Append3 := InternalAppend(destinationString, sources);
END_METHOD

METHOD Append4 : BOOL
VAR_INPUT
	destinationString : ANY_STRING;
	sourceString1 : WSTRING(255);
	sourceString2 : WSTRING(255);
	sourceString3 : WSTRING(255);
	sourceString4 : WSTRING(255);
END_VAR
VAR
	sources : ARRAY [1..4] OF POINTER TO WSTRING(255);
END_VAR
sources[1] := ADR(sourceString1);
sources[2] := ADR(sourceString2);
sources[3] := ADR(sourceString3);
sources[4] := ADR(sourceString4);

Append4 := InternalAppend(destinationString, sources);
END_METHOD

METHOD Append5 : BOOL
VAR_INPUT
	destinationString : ANY_STRING;
	sourceString1 : WSTRING(255);
	sourceString2 : WSTRING(255);
	sourceString3 : WSTRING(255);
	sourceString4 : WSTRING(255);
	sourceString5 : WSTRING(255);
END_VAR
VAR
	sources : ARRAY [1..5] OF POINTER TO WSTRING(255);
END_VAR
sources[1] := ADR(sourceString1);
sources[2] := ADR(sourceString2);
sources[3] := ADR(sourceString3);
sources[4] := ADR(sourceString4);
sources[5] := ADR(sourceString5);

Append5 := InternalAppend(destinationString, sources);
END_METHOD

METHOD Append6 : BOOL
VAR_INPUT
	destinationString : ANY_STRING;
	sourceString1 : WSTRING(255);
	sourceString2 : WSTRING(255);
	sourceString3 : WSTRING(255);
	sourceString4 : WSTRING(255);
	sourceString5 : WSTRING(255);
	sourceString6 : WSTRING(255);
END_VAR
VAR
	sources : ARRAY [1..6] OF POINTER TO WSTRING(255);
END_VAR
sources[1] := ADR(sourceString1);
sources[2] := ADR(sourceString2);
sources[3] := ADR(sourceString3);
sources[4] := ADR(sourceString4);
sources[5] := ADR(sourceString5);
sources[6] := ADR(sourceString6);

Append6 := InternalAppend(destinationString, sources);
END_METHOD

METHOD Append7 : BOOL
VAR_INPUT
	destinationString : ANY_STRING;
	sourceString1 : WSTRING(255);
	sourceString2 : WSTRING(255);
	sourceString3 : WSTRING(255);
	sourceString4 : WSTRING(255);
	sourceString5 : WSTRING(255);
	sourceString6 : WSTRING(255);
	sourceString7 : WSTRING(255);
END_VAR
VAR
	sources : ARRAY [1..7] OF POINTER TO WSTRING(255);
END_VAR
sources[1] := ADR(sourceString1);
sources[2] := ADR(sourceString2);
sources[3] := ADR(sourceString3);
sources[4] := ADR(sourceString4);
sources[5] := ADR(sourceString5);
sources[6] := ADR(sourceString6);
sources[7] := ADR(sourceString7);

Append7 := InternalAppend(destinationString, sources);
END_METHOD

METHOD Append8 : BOOL
VAR_INPUT
	destinationString : ANY_STRING;
	sourceString1 : WSTRING(255);
	sourceString2 : WSTRING(255);
	sourceString3 : WSTRING(255);
	sourceString4 : WSTRING(255);
	sourceString5 : WSTRING(255);
	sourceString6 : WSTRING(255);
	sourceString7 : WSTRING(255);
	sourceString8 : WSTRING(255);
END_VAR
VAR
	sources : ARRAY [1..8] OF POINTER TO WSTRING(255);
END_VAR
sources[1] := ADR(sourceString1);
sources[2] := ADR(sourceString2);
sources[3] := ADR(sourceString3);
sources[4] := ADR(sourceString4);
sources[5] := ADR(sourceString5);
sources[6] := ADR(sourceString6);
sources[7] := ADR(sourceString7);
sources[8] := ADR(sourceString8);

Append8 := InternalAppend(destinationString, sources);
END_METHOD

METHOD Append9 : BOOL
VAR_INPUT
	destinationString : ANY_STRING;
	sourceString1 : WSTRING(255);
	sourceString2 : WSTRING(255);
	sourceString3 : WSTRING(255);
	sourceString4 : WSTRING(255);
	sourceString5 : WSTRING(255);
	sourceString6 : WSTRING(255);
	sourceString7 : WSTRING(255);
	sourceString8 : WSTRING(255);
	sourceString9 : WSTRING(255);
END_VAR
VAR
	sources : ARRAY [1..9] OF POINTER TO WSTRING(255);
END_VAR
sources[1] := ADR(sourceString1);
sources[2] := ADR(sourceString2);
sources[3] := ADR(sourceString3);
sources[4] := ADR(sourceString4);
sources[5] := ADR(sourceString5);
sources[6] := ADR(sourceString6);
sources[7] := ADR(sourceString7);
sources[8] := ADR(sourceString8);
sources[9] := ADR(sourceString9);

Append9 := InternalAppend(destinationString, sources);
END_METHOD

METHOD Concat10 : WSTRING(255)
VAR_INPUT
	string1 : WSTRING(255);
	string2 : WSTRING(255);
	string3 : WSTRING(255);
	string4 : WSTRING(255);
	string5 : WSTRING(255);
	string6 : WSTRING(255);
	string7 : WSTRING(255);
	string8 : WSTRING(255);
	string9 : WSTRING(255);
	string10 : WSTRING(255);
END_VAR
Concat10 := Tc2_Standard.WCONCAT(
	Tc2_Standard.WCONCAT(
		Tc2_Standard.WCONCAT(Tc2_Standard.WCONCAT(string1, string2), Tc2_Standard.WCONCAT(string3, string4)), 
		Tc2_Standard.WCONCAT(Tc2_Standard.WCONCAT(string5, string6), Tc2_Standard.WCONCAT(string7, string8)) 
	),
	Tc2_Standard.WCONCAT(string9, string10));
END_METHOD

METHOD Concat11 : WSTRING(255)
VAR_INPUT
	string1 : WSTRING(255);
	string2 : WSTRING(255);
	string3 : WSTRING(255);
	string4 : WSTRING(255);
	string5 : WSTRING(255);
	string6 : WSTRING(255);
	string7 : WSTRING(255);
	string8 : WSTRING(255);
	string9 : WSTRING(255);
	string10 : WSTRING(255);
	string11 : WSTRING(255);
END_VAR
Concat11 := Tc2_Standard.WCONCAT(
	Tc2_Standard.WCONCAT(
		Tc2_Standard.WCONCAT(Tc2_Standard.WCONCAT(string1, string2), Tc2_Standard.WCONCAT(string3, string4)), 
		Tc2_Standard.WCONCAT(Tc2_Standard.WCONCAT(string5, string6), Tc2_Standard.WCONCAT(string7, string8)) 
	),
	Tc2_Standard.WCONCAT(
		Tc2_Standard.WCONCAT(string9, string10),
		string11
	)
);
END_METHOD

METHOD Concat12 : WSTRING(255)
VAR_INPUT
	string1 : WSTRING(255);
	string2 : WSTRING(255);
	string3 : WSTRING(255);
	string4 : WSTRING(255);
	string5 : WSTRING(255);
	string6 : WSTRING(255);
	string7 : WSTRING(255);
	string8 : WSTRING(255);
	string9 : WSTRING(255);
	string10 : WSTRING(255);
	string11 : WSTRING(255);
	string12 : WSTRING(255);
END_VAR
Concat12 := Tc2_Standard.WCONCAT(
	Tc2_Standard.WCONCAT(
		Tc2_Standard.WCONCAT(Tc2_Standard.WCONCAT(string1, string2), Tc2_Standard.WCONCAT(string3, string4)), 
		Tc2_Standard.WCONCAT(Tc2_Standard.WCONCAT(string5, string6), Tc2_Standard.WCONCAT(string7, string8)) 
	),
	Tc2_Standard.WCONCAT(
		Tc2_Standard.WCONCAT(string9, string10),
		Tc2_Standard.WCONCAT(string11, string12)
	)
);
END_METHOD

METHOD Concat13 : WSTRING(255)
VAR_INPUT
	string1 : WSTRING(255);
	string2 : WSTRING(255);
	string3 : WSTRING(255);
	string4 : WSTRING(255);
	string5 : WSTRING(255);
	string6 : WSTRING(255);
	string7 : WSTRING(255);
	string8 : WSTRING(255);
	string9 : WSTRING(255);
	string10 : WSTRING(255);
	string11 : WSTRING(255);
	string12 : WSTRING(255);
	string13 : WSTRING(255);
END_VAR
Concat13 := Tc2_Standard.WCONCAT(
	Tc2_Standard.WCONCAT(
		Tc2_Standard.WCONCAT(Tc2_Standard.WCONCAT(string1, string2), Tc2_Standard.WCONCAT(string3, string4)), 
		Tc2_Standard.WCONCAT(Tc2_Standard.WCONCAT(string5, string6), Tc2_Standard.WCONCAT(string7, string8)) 
	),
	Tc2_Standard.WCONCAT(
		Tc2_Standard.WCONCAT(Tc2_Standard.WCONCAT(string9, string10), Tc2_Standard.WCONCAT(string11, string12)),
		string13
	)
);
END_METHOD

METHOD Concat14 : WSTRING(255)
VAR_INPUT
	string1 : WSTRING(255);
	string2 : WSTRING(255);
	string3 : WSTRING(255);
	string4 : WSTRING(255);
	string5 : WSTRING(255);
	string6 : WSTRING(255);
	string7 : WSTRING(255);
	string8 : WSTRING(255);
	string9 : WSTRING(255);
	string10 : WSTRING(255);
	string11 : WSTRING(255);
	string12 : WSTRING(255);
	string13 : WSTRING(255);
	string14 : WSTRING(255);
END_VAR
Concat14 := Tc2_Standard.WCONCAT(
	Tc2_Standard.WCONCAT(
		Tc2_Standard.WCONCAT(Tc2_Standard.WCONCAT(string1, string2), Tc2_Standard.WCONCAT(string3, string4)), 
		Tc2_Standard.WCONCAT(Tc2_Standard.WCONCAT(string5, string6), Tc2_Standard.WCONCAT(string7, string8)) 
	),
	Tc2_Standard.WCONCAT(
		Tc2_Standard.WCONCAT(Tc2_Standard.WCONCAT(string9, string10), Tc2_Standard.WCONCAT(string11, string12)),
		Tc2_Standard.WCONCAT(string13, string14)
	)
);
END_METHOD

METHOD Concat2 : WSTRING(255)
VAR_INPUT
	string1 : WSTRING(255);
	string2 : WSTRING(255);
END_VAR
Concat2 := Tc2_Standard.WCONCAT(string1, string2);
END_METHOD

METHOD Concat3 : WSTRING(255)
VAR_INPUT
	string1 : WSTRING(255);
	string2 : WSTRING(255);
	string3 : WSTRING(255);
END_VAR
Concat3 := Tc2_Standard.WCONCAT(Tc2_Standard.WCONCAT(string1, string2), string3);
END_METHOD

METHOD Concat4 : WSTRING(255)
VAR_INPUT
	string1 : WSTRING(255);
	string2 : WSTRING(255);
	string3 : WSTRING(255);
	string4 : WSTRING(255);
END_VAR
Concat4 := Tc2_Standard.WCONCAT(Tc2_Standard.WCONCAT(string1, string2), Tc2_Standard.WCONCAT(string3, string4));
END_METHOD

METHOD Concat5 : WSTRING(255)
VAR_INPUT
	string1 : WSTRING(255);
	string2 : WSTRING(255);
	string3 : WSTRING(255);
	string4 : WSTRING(255);
	string5 : WSTRING(255);
END_VAR
Concat5 := Tc2_Standard.WCONCAT(Tc2_Standard.WCONCAT(Tc2_Standard.WCONCAT(string1, string2), Tc2_Standard.WCONCAT(string3, string4)), string5);
END_METHOD

METHOD Concat6 : WSTRING(255)
VAR_INPUT
	string1 : WSTRING(255);
	string2 : WSTRING(255);
	string3 : WSTRING(255);
	string4 : WSTRING(255);
	string5 : WSTRING(255);
	string6 : WSTRING(255);
END_VAR
Concat6 := Tc2_Standard.WCONCAT(
	Tc2_Standard.WCONCAT(Tc2_Standard.WCONCAT(string1, string2), Tc2_Standard.WCONCAT(string3, string4)), 
	Tc2_Standard.WCONCAT(string5, string6)
);
END_METHOD

METHOD Concat7 : WSTRING(255)
VAR_INPUT
	string1 : WSTRING(255);
	string2 : WSTRING(255);
	string3 : WSTRING(255);
	string4 : WSTRING(255);
	string5 : WSTRING(255);
	string6 : WSTRING(255);
	string7 : WSTRING(255);
END_VAR
Concat7 := Tc2_Standard.WCONCAT(
	Tc2_Standard.WCONCAT(Tc2_Standard.WCONCAT(string1, string2), Tc2_Standard.WCONCAT(string3, string4)), 
	Tc2_Standard.WCONCAT(Tc2_Standard.WCONCAT(string5, string6), string7)
);
END_METHOD

METHOD Concat8 : WSTRING(255)
VAR_INPUT
	string1 : WSTRING(255);
	string2 : WSTRING(255);
	string3 : WSTRING(255);
	string4 : WSTRING(255);
	string5 : WSTRING(255);
	string6 : WSTRING(255);
	string7 : WSTRING(255);
	string8 : WSTRING(255);
END_VAR
Concat8 := Tc2_Standard.WCONCAT(
	Tc2_Standard.WCONCAT(Tc2_Standard.WCONCAT(string1, string2), Tc2_Standard.WCONCAT(string3, string4)), 
	Tc2_Standard.WCONCAT(Tc2_Standard.WCONCAT(string5, string6), Tc2_Standard.WCONCAT(string7, string8)) 
);
END_METHOD

METHOD Concat9 : WSTRING(255)
VAR_INPUT
	string1 : WSTRING(255);
	string2 : WSTRING(255);
	string3 : WSTRING(255);
	string4 : WSTRING(255);
	string5 : WSTRING(255);
	string6 : WSTRING(255);
	string7 : WSTRING(255);
	string8 : WSTRING(255);
	string9 : WSTRING(255);
END_VAR
Concat9 := Tc2_Standard.WCONCAT(
	Tc2_Standard.WCONCAT(
		Tc2_Standard.WCONCAT(Tc2_Standard.WCONCAT(string1, string2), Tc2_Standard.WCONCAT(string3, string4)), 
		Tc2_Standard.WCONCAT(Tc2_Standard.WCONCAT(string5, string6), Tc2_Standard.WCONCAT(string7, string8)) 
	),
	string9);
END_METHOD

METHOD DateAndTimeToString : WSTRING
VAR_INPUT
	value : DATE_AND_TIME;
	dateValuesSeparator : STRING(1) := '_';
	dateAndTimeSeparator : STRING(1) := '-';
	timeValuesSeparator : STRING(1) := '_';
END_VAR
VAR
	result : STRING;
END_VAR
result := TO_STRING(value);

result := Tc2_Standard.DELETE(result, 3, 1);

result := Tc2_Standard.REPLACE(result, dateValuesSeparator, 1, 5);
result := Tc2_Standard.REPLACE(result, dateValuesSeparator, 1, 8);
result := Tc2_Standard.REPLACE(result, dateAndTimeSeparator, 1, 11);
result := Tc2_Standard.REPLACE(result, timeValuesSeparator, 1, 14);
result := Tc2_Standard.REPLACE(result, timeValuesSeparator, 1, 17);

DateAndTimeToString := TO_WSTRING(result);
END_METHOD

METHOD INTERNAL InternalAnyToString : WSTRING(255)
VAR_INPUT
	value : __System.AnyType;
END_VAR
VAR
	anyBool : POINTER TO BOOL;

	anyByte : POINTER TO BYTE;
	anyWord : POINTER TO WORD;
	anyDWord : POINTER TO LWORD;
	anyLWord : POINTER TO LWORD;
	
	anySInt : POINTER TO SINT;
	anyInt : POINTER TO INT;
	anyDInt : POINTER TO DINT;
	anyLInt : POINTER TO LINT;
	
	anyUSInt : POINTER TO USINT;
	anyUInt : POINTER TO UINT;
	anyUDInt : POINTER TO UDINT;
	anyULInt : POINTER TO ULINT;
	
	anyReal : POINTER TO REAL;
	anyLReal : POINTER TO LREAL;

	anyString : POINTER TO STRING(255);
	anyWString : POINTER TO WSTRING(255);
	
	anyTime : POINTER TO TIME;
	anyLTime : POINTER TO LTIME;
	anyDate : POINTER TO DATE;
	anyDateAndTime : POINTER TO DATE_AND_TIME;
	anyTimeOfDay : POINTER TO TOD;
END_VAR
CASE value.TypeClass OF
	__SYSTEM.TYPE_CLASS.TYPE_BOOL:
		anyBool := value.pValue;
		InternalAnyToString := TO_WSTRING(anyBool^);		
	
	__SYSTEM.TYPE_CLASS.TYPE_BIT:
		anyByte := value.pValue;
		IF anyByte^ > 0 THEN
			InternalAnyToString := "1";		
		ELSE
			InternalAnyToString := "0";		
		END_IF
	
	__SYSTEM.TYPE_CLASS.TYPE_BYTE:
		anyByte := value.pValue;
		InternalAnyToString := TO_WSTRING(anyByte^);		
	__SYSTEM.TYPE_CLASS.TYPE_WORD:
		anyWord := value.pValue;
		InternalAnyToString := TO_WSTRING(anyWord^);
	__SYSTEM.TYPE_CLASS.TYPE_DWORD:
		anyDWord := value.pValue;
		InternalAnyToString := TO_WSTRING(anyDWord^);
	__SYSTEM.TYPE_CLASS.TYPE_LWORD:
		anyLWord := value.pValue;
		InternalAnyToString := TO_WSTRING(anyLWord^);
		
	__SYSTEM.TYPE_CLASS.TYPE_SINT:
		anySInt := value.pValue;
		InternalAnyToString := TO_WSTRING(anySInt^);
	__SYSTEM.TYPE_CLASS.TYPE_INT:
		anyInt := value.pValue;
		InternalAnyToString := TO_WSTRING(anyInt^);		
	__SYSTEM.TYPE_CLASS.TYPE_DINT:
		anyDInt := value.pValue;
		InternalAnyToString := TO_WSTRING(anyDInt^);
	__SYSTEM.TYPE_CLASS.TYPE_LINT:
		anyLInt := value.pValue;
		InternalAnyToString := TO_WSTRING(anyLInt^);
		
	__SYSTEM.TYPE_CLASS.TYPE_USINT:
		anyUSInt := value.pValue;
		InternalAnyToString := TO_WSTRING(anyUSInt^);
	__SYSTEM.TYPE_CLASS.TYPE_UINT:
		anyUInt := value.pValue;
		InternalAnyToString := TO_WSTRING(anyUInt^);		
	__SYSTEM.TYPE_CLASS.TYPE_UDINT:
		anyUDInt := value.pValue;
		InternalAnyToString := TO_WSTRING(anyUDInt^);
	__SYSTEM.TYPE_CLASS.TYPE_ULINT:
		anyULInt := value.pValue;
		InternalAnyToString := TO_WSTRING(anyULInt^);

	__SYSTEM.TYPE_CLASS.TYPE_REAL:
		anyReal := value.pValue;
		InternalAnyToString := TO_WSTRING(anyReal^);
	__SYSTEM.TYPE_CLASS.TYPE_LREAL:
		anyLReal := value.pValue;
		InternalAnyToString := TO_WSTRING(anyLReal^);
	
	__SYSTEM.TYPE_CLASS.TYPE_STRING:
		anyString := value.pValue;
		InternalAnyToString := TO_WSTRING(anyString^);
	__SYSTEM.TYPE_CLASS.TYPE_WSTRING:
		anyWString := value.pValue;
		InternalAnyToString := anyWString^;
	
	__SYSTEM.TYPE_CLASS.TYPE_TIME:
		anyTime := value.pValue;
		InternalAnyToString := TO_WSTRING(anyTime^);
	__SYSTEM.TYPE_CLASS.TYPE_LTIME:
		anyLTime := value.pValue;
		InternalAnyToString := TO_WSTRING(anyLTime^);
	__SYSTEM.TYPE_CLASS.TYPE_DATE:
		anyDate := value.pValue;
		InternalAnyToString := TO_WSTRING(anyDate^);
	__SYSTEM.TYPE_CLASS.TYPE_DATEANDTIME:
		anyDateAndTime := value.pValue;
		InternalAnyToString := TO_WSTRING(anyDateAndTime^);  
	__SYSTEM.TYPE_CLASS.TYPE_TIMEOFDAY:
		anyTimeOfDay := value.pValue;
		InternalAnyToString := TO_WSTRING(anyTimeOfDay^);
	
	__SYSTEM.TYPE_CLASS.TYPE_POINTER, __SYSTEM.TYPE_CLASS.TYPE_REFERENCE:
		InternalAnyToString := TO_WSTRING(Tc2_Utilities.PVOID_TO_HEXSTR(anyDate, 8, FALSE));		
	
	(*__SYSTEM.TYPE_CLASS.TYPE_SUBRANGE:
	__SYSTEM.TYPE_CLASS.TYPE_ENUM:
	__SYSTEM.TYPE_CLASS.TYPE_ARRAY:
	__SYSTEM.TYPE_CLASS.TYPE_PARAMS:
	__SYSTEM.TYPE_CLASS.TYPE_USERDEF:
	__SYSTEM.TYPE_CLASS.TYPE_NONE:
	__SYSTEM.TYPE_CLASS.TYPE_ANY:
	__SYSTEM.TYPE_CLASS.TYPE_ANYBIT:
	__SYSTEM.TYPE_CLASS.TYPE_ANYDATE:
	__SYSTEM.TYPE_CLASS.TYPE_ANYINT:
	__SYSTEM.TYPE_CLASS.TYPE_ANYNUM:
	__SYSTEM.TYPE_CLASS.TYPE_ANYREAL:
	__SYSTEM.TYPE_CLASS.TYPE_LAZY:
	__SYSTEM.TYPE_CLASS.TYPE_BITCONST:*)
	ELSE
		IF value.pValue <> 0 THEN
			InternalAnyToString := TO_WSTRING(value.pValue^); 
		ELSE
			InternalAnyToString := "NULL";
		END_IF
END_CASE
END_METHOD

METHOD INTERNAL InternalAppend : BOOL
VAR_INPUT
	destinationString : __SYSTEM.AnyType;
END_VAR
VAR_IN_OUT
	sourceStrings : ARRAY [*] OF POINTER TO WSTRING(255);
END_VAR
VAR
	i : DINT;
END_VAR
IF destinationString.TypeClass <> __SYSTEM.TYPE_CLASS.TYPE_WSTRING THEN
	RETURN;
END_IF	

FOR i := LOWER_BOUND(sourceStrings, 1) TO UPPER_BOUND(sourceStrings, 1) DO
	InternalAppend := Tc2_Utilities.WCONCAT2(destinationString.pValue, sourceStrings[i], destinationString.pValue, TO_UDINT(destinationString.diSize));	
END_FOR
END_METHOD

END_PROGRAM

// ---- Exceptions/General/ArgumentOutOfRange/ArgumentOutOfRangeException.TcPOU
{attribute 'enable_dynamic_creation'}	
{attribute 'no_explicit_call' := 'do not call this function block directly'} 
FUNCTION_BLOCK ArgumentOutOfRangeException EXTENDS GeneralException
VAR
	_ClassName : STRING := __POUNAME();
END_VAR

{attribute 'monitoring' := 'call'}
PROPERTY ClassName : STRING
GET
ClassName := _ClassName;
END_GET
END_PROPERTY

METHOD Clone : IObject
VAR
	exceptionClone : POINTER TO ArgumentOutOfRangeException;
END_VAR
exceptionClone := __NEW(ArgumentOutOfRangeException);

Clone := InternalClone(exceptionClone);
END_METHOD

METHOD Throw
VAR_INPUT
	sourceNamespaceName : STRING;
	sourceClassName : STRING;
	sourceMethodName : STRING;
	sourcePosition : STRING;
	argumentName : STRING;
	argumentValue : ANY;
	fatal : BOOL := FALSE;
END_VAR
VAR
	valueAsString : WSTRING(255);
	stringBuilder : WideStringBuilder;
	message : ERROR_MESSAGE;
	zeroErrorCode : UDINT;
	nullInnerException : REFERENCE TO Exception REF= 0;
END_VAR
valueAsString := WideStringHelper.InternalAnyToString(argumentValue);

stringBuilder
	.AppendString("Argument '")
	.Append(argumentName)
	.AppendString("' has invalid value '")
	.AppendString(valueAsString)
	.AppendString("in method or function '");

AppendProgramOrganizationUnitFullName(stringBuilder);

stringBuilder
	.AppendString("'")
	.AssignToString(message);

InternalThrow(sourceNamespaceName, sourceClassName, sourceMethodName, sourcePosition, message, zeroErrorCode, fatal, nullInnerException);
END_METHOD

END_FUNCTION_BLOCK

// ---- Exceptions/General/GeneralException.TcPOU
{attribute 'enable_dynamic_creation'}	
{attribute 'no_explicit_call' := 'do not call this function block directly'} 
FUNCTION_BLOCK ABSTRACT GeneralException EXTENDS Exception
VAR_OUTPUT
	ErrorCode : UDINT;
	
	InnerException : POINTER TO Exception;
END_VAR
VAR
	_Message : ERROR_MESSAGE;
END_VAR

{attribute 'monitoring' := 'call'}
PROPERTY Empty : BOOL
GET
Empty := ErrorCode = 0 AND_THEN _Message = "";
END_GET
END_PROPERTY

METHOD FB_exit : BOOL
VAR_INPUT
	(* if TRUE, the exit method is called for exiting an instance that is copied afterwards (online change).*)
	bInCopyCode	: BOOL;
END_VAR
IF InnerException <> 0 THEN 
	__DELETE(InnerException);
END_IF
END_METHOD

METHOD GetMessage : ERROR_MESSAGE
VAR_INPUT
	showTimestamp : BOOL := FALSE;
	showSource : BOOL := FALSE;
END_VAR
VAR
	stringBuilder : WideStringBuilder;

	innerExceptionMessage : ERROR_MESSAGE;
END_VAR
stringBuilder
	.Append(_Message)
	.AppendStringIf(ERROR_CODE_PREFIX, ErrorCode > 0)
	.AppendIf(ErrorCode, ErrorCode > 0);	

IF showTimestamp THEN
	stringBuilder.AppendString(TIME_PREFIX);
	AppendTimestampDescription(stringBuilder);
END_IF

IF showSource THEN
	stringBuilder.AppendString(SOURCE_PREFIX);
	AppendSourceDescription(stringBuilder);
END_IF

IF InnerException <> 0 THEN
	innerExceptionMessage := InnerException^.GetMessage(showTimestamp, showSource);
END_IF

IF innerExceptionMessage <> "" THEN
	stringBuilder
		.AppendString(INNER_MESSAGE_PREFIX)
		.AppendString(innerExceptionMessage);	
END_IF

stringBuilder.AssignToString(GetMessage);
END_METHOD

METHOD PROTECTED InternalClone : IObject
VAR_INPUT
	exceptionClone : POINTER TO GeneralException;
END_VAR
VAR
	innerExceptionClone : IObject;
END_VAR
exceptionClone^.ErrorCode := ErrorCode;
exceptionClone^._Message := _Message;
exceptionClone^.Fatal := Fatal;
exceptionClone^.SourceNamespaceName := SourceNamespaceName;
exceptionClone^.SourceClassName := SourceClassName;
exceptionClone^.SourceMethodName := SourceMethodName;
exceptionClone^.SourcePosition := SourcePosition;
exceptionClone^.LocalTimestamp := LocalTimestamp;	
exceptionClone^.UtcTimestamp := UtcTimestamp;	

IF InnerException <> 0 THEN
	innerExceptionClone := InnerException^.Clone(); 
	__QUERYPOINTER(innerExceptionClone, exceptionClone^.InnerException);
END_IF

InternalClone := exceptionClone^;
END_METHOD

METHOD PROTECTED InternalThrow
VAR_IN_OUT CONSTANT
	sourceNamespaceName : STRING;
	sourceClassName : STRING;
	sourceMethodName : STRING;
	sourcePosition : STRING;
	message : ERROR_MESSAGE;
	errorCode : UDINT;
	fatal : BOOL;
	innerException : Exception;
END_VAR
THIS^.SourceNamespaceName := sourceNamespaceName;	
THIS^.SourceClassName := sourceClassName;
THIS^.SourceMethodName := SEL(Tc2_Standard.FIND(sourceMethodName, sourceClassName) <> 1, Tc2_Standard.DELETE(sourceMethodName, Tc2_Standard.LEN(sourceClassName) + 1, 1), sourceMethodName); 
THIS^.SourcePosition := sourcePosition;
THIS^._Message := message;
THIS^.ErrorCode := errorCode;
THIS^.Fatal := fatal;
THIS^.LocalTimestamp := SystemDateTimeManager.SystemLocalDateTime;
THIS^.UtcTimestamp := SystemDateTimeManager.SystemUtcDateTime;

IF __ISVALIDREF(innerException) THEN
	THIS^.InnerException := ADR(innerException);
ELSE
	THIS^.InnerException := 0;
END_IF

ExceptionManager.Throw(THIS^);
END_METHOD

END_FUNCTION_BLOCK

// ---- Primitives/DateAndTime/SystemDateTimeManager.TcPOU
{attribute 'no_explicit_call' := 'do not call this function block directly'} 
PROGRAM SystemDateTimeManager
VAR_OUTPUT
	{attribute 'OPC.UA.DA.Access' := '1'}
	MinDateTime : DATE_AND_TIME := DT#1970-01-01-00:00;
	
	{attribute 'OPC.UA.DA.Access' := '1'}
	SystemTimeZoneId : Tc2_Utilities.E_TimeZoneID;
	{attribute 'OPC.UA.DA.Access' := '1'}
	SystemTimeZoneInformation : Tc2_Utilities.ST_TimeZoneInformation;
	{attribute 'OPC.UA.DA.Access' := '1'}	
	SystemTimeZoneValid : BOOL;
	
	{attribute 'OPC.UA.DA.Access' := '1'}	
	SystemLocalDateTime : DATE_AND_TIME;
	{attribute 'OPC.UA.DA.Access' := '1'}	
	SystemLocalDate : DATE;
	{attribute 'OPC.UA.DA.Access' := '1'}	
	SystemLocalTime : TIME;
	{attribute 'OPC.UA.DA.Access' := '1'}	
	SystemLocalTimeOfDay : TIME_OF_DAY;
	
	{attribute 'OPC.UA.DA.Access' := '1'}	
	SystemUtcDateTime : DATE_AND_TIME;
	{attribute 'OPC.UA.DA.Access' := '1'}	
	SystemUtcDate : DATE;
	{attribute 'OPC.UA.DA.Access' := '1'}	
	SystemUtcTime : TIME;
	{attribute 'OPC.UA.DA.Access' := '1'}	
	SystemUtcTimeOfDay : TIME_OF_DAY;

	{attribute 'OPC.UA.DA.Access' := '1'}	
	SystemFileTime : Tc2_Utilities.T_FILETIME;
	{attribute 'OPC.UA.DA.Access' := '1'}	
	SystemFileTime64 : Tc2_Utilities.T_FILETIME64;
END_VAR
VAR
	{attribute 'OPC.UA.DA' := '0'}
	_LocalSystemTime : Tc2_Utilities.FB_LocalSystemTime; 
	{attribute 'OPC.UA.DA' := '0'}
	_GetTimeZone : Tc2_Utilities.FB_GetTimeZoneInformation;
	{attribute 'OPC.UA.DA' := '0'}	
	_LocalTimeToUtcTime : FB_TzSpecificLocalTimeToSystemTime;
END_VAR

METHOD Execute : BOOL
IF SystemTimeZoneId = Tc2_Utilities.E_TimeZoneID.eTimeZoneID_Unknown OR_ELSE SystemTimeZoneId = Tc2_Utilities.E_TimeZoneID.eTimeZoneID_Invalid THEN
	_GetTimeZone(bExecute := TRUE, tTimeout := T#1S);
	
	IF _GetTimeZone.bError THEN
		_GetTimeZone(bExecute := FALSE);
		_GetTimeZone(bExecute := TRUE);
	ELSE
		SystemTimeZoneId := _GetTimeZone.tzID;
		SystemTimeZoneInformation := _GetTimeZone.tzInfo;
		SystemTimeZoneValid := TRUE; 
	END_IF
END_IF

_LocalSystemTime(bEnable := TRUE);

IF SystemTimeZoneValid THEN	
	SystemLocalDateTime := Tc2_Utilities.SYSTEMTIME_TO_DT(_LocalSystemTime.systemTime);
	SystemLocalDate := DT_TO_DATE(SystemLocalDateTime);
	SystemLocalTime := TO_TIME(StringHelper.Concat9('T#', TO_STRING(_LocalSystemTime.systemTime.wHour), 'h', TO_STRING(_LocalSystemTime.systemTime.wMinute), 'm', TO_STRING(_LocalSystemTime.systemTime.wSecond), 's', TO_STRING(_LocalSystemTime.systemTime.wMilliseconds), 'ms'));	
	SystemLocalTimeOfDay := TO_TOD(StringHelper.Concat8('TOD#', TO_STRING(_LocalSystemTime.systemTime.wHour), ':', TO_STRING(_LocalSystemTime.systemTime.wMinute), ':', TO_STRING(_LocalSystemTime.systemTime.wSecond), '.', TO_STRING(_LocalSystemTime.systemTime.wMilliseconds)));	

	_LocalTimeToUtcTime(in := _LocalSystemTime.systemTime, tzInfo := _GetTimeZone.tzInfo);	

	SystemUtcDateTime := Tc2_Utilities.SYSTEMTIME_TO_DT(_LocalTimeToUtcTime.out);
	SystemUtcDate := DT_TO_DATE(SystemUtcDateTime);
	SystemUtcTime := TO_TIME(StringHelper.Concat9('T#', TO_STRING(_LocalTimeToUtcTime.out.wHour), 'h', TO_STRING(_LocalTimeToUtcTime.out.wMinute), 'm', TO_STRING(_LocalTimeToUtcTime.out.wSecond), 's', TO_STRING(_LocalTimeToUtcTime.out.wMilliseconds), 'ms'));	
	SystemUtcTimeOfDay := TO_TOD(StringHelper.Concat8('TOD#', TO_STRING(_LocalTimeToUtcTime.out.wHour), ':', TO_STRING(_LocalTimeToUtcTime.out.wMinute), ':', TO_STRING(_LocalTimeToUtcTime.out.wSecond), '.', TO_STRING(_LocalTimeToUtcTime.out.wMilliseconds)));	

	SystemFileTime := Tc2_Utilities.SYSTEMTIME_TO_FILETIME(_LocalSystemTime.systemTime);
	SystemFileTime64 := Tc2_Utilities.SYSTEMTIME_TO_FILETIME64(_LocalSystemTime.systemTime);
END_IF
END_METHOD

PROPERTY SystemTime : TIMESTRUCT
GET
SystemTime := _LocalSystemTime.systemTime;
END_GET
END_PROPERTY

{attribute 'OPC.UA.DA.Property' := '1'}
{attribute 'monitoring' := 'call'}
PROPERTY SystemTimeSynchronisationInterval : DWORD
GET
SystemTimeSynchronisationInterval := _LocalSystemTime.dwCycle;
END_GET
SET
_LocalSystemTime.dwCycle := SystemTimeSynchronisationInterval;
END_SET
END_PROPERTY

PROPERTY SystemTimeValid : BOOL
GET
SystemTimeValid := SystemTimeZoneValid AND_THEN _LocalSystemTime.bValid;
END_GET
END_PROPERTY

END_PROGRAM

// ---- Exceptions/ExceptionManager.TcPOU
{attribute 'no_explicit_call' := 'do not call this function block directly'} 
PROGRAM ExceptionManager
VAR
	_Exception : POINTER TO Exception;
	_EmptyException : EmptyException;
	_SystemException : SystemException;	
END_VAR

METHOD Cleanup
IF _Exception <> 0 THEN
	__DELETE(_Exception);		
END_IF
END_METHOD

// Result is always not null. Returns EmptyException instance by default
METHOD GetLastException : IException
VAR_IN_OUT CONSTANT 
	exceptionCode : __SYSTEM.ExceptionCode;
END_VAR
IF exceptionCode = __SYSTEM.ExceptionCode.RTSEXCPT_DIVIDEBYZERO AND_THEN _Exception <> 0 THEN
	GetLastException := _Exception^;
ELSE
	_SystemException.SetExceptionCode(exceptionCode);
	GetLastException := _SystemException;
END_IF
END_METHOD

METHOD Throw
VAR_INPUT
	exception : IException;
END_VAR
VAR
	fakeVariable : INT := 0;
	exceptionCloneInterface : IObject;
END_VAR
IF _Exception <> 0 THEN
	__DELETE(_Exception);
END_IF

__QUERYPOINTER(exception.Clone(), _Exception);

// fake devision by zero
fakeVariable := fakeVariable / fakeVariable;
END_METHOD

END_PROGRAM

// ---- Exceptions/Empty/EmptyException.TcPOU
{attribute 'enable_dynamic_creation'}	
{attribute 'no_explicit_call' := 'do not call this function block directly'} 
FUNCTION_BLOCK EmptyException EXTENDS Exception
VAR
	_ClassName : STRING := __POUNAME();
END_VAR

{attribute 'monitoring' := 'call'}
PROPERTY ClassName : STRING
GET
ClassName := _ClassName;
END_GET
END_PROPERTY

METHOD Clone : IObject
VAR
	exceptionClone : POINTER TO EmptyException;
END_VAR
exceptionClone := __NEW(EmptyException);

Clone := exceptionClone^;
END_METHOD

{attribute 'monitoring' := 'call'}
PROPERTY Empty : BOOL
GET
Empty := TRUE;
END_GET
END_PROPERTY

METHOD GetMessage : ERROR_MESSAGE
VAR_INPUT
	showTimestamp : BOOL := FALSE;
	showSource : BOOL := FALSE;
END_VAR
GetMessage := "";
END_METHOD

END_FUNCTION_BLOCK

// ---- Exceptions/System/SystemException.TcPOU
{attribute 'enable_dynamic_creation'}	
{attribute 'no_explicit_call' := 'do not call this function block directly'} 
FUNCTION_BLOCK SystemException EXTENDS Exception
VAR_OUTPUT
	ExceptionCode : __SYSTEM.ExceptionCode;
END_VAR
VAR
	_ClassName : STRING := __POUNAME();
END_VAR
VAR CONSTANT
	SYSTEM_EXCEPTION_PREFIX : WSTRING(16) := "System exception";
END_VAR

{attribute 'monitoring' := 'call'}
PROPERTY ClassName : STRING
GET
ClassName := _ClassName;
END_GET
END_PROPERTY

METHOD Clone : IObject
VAR
	exceptionClone : POINTER TO SystemException;
END_VAR
exceptionClone := __NEW(SystemException);

exceptionClone^.ExceptionCode := ExceptionCode;
exceptionClone^.LocalTimestamp := LocalTimestamp;
exceptionClone^.UtcTimestamp := UtcTimestamp;

Clone := exceptionClone^;
END_METHOD

{attribute 'monitoring' := 'call'}
PROPERTY Empty : BOOL
GET
Empty := TRUE;
END_GET
END_PROPERTY

METHOD FB_init : BOOL
VAR_INPUT
	(* if TRUE, the retain variables are initialized (warm start / cold start)*)
	bInitRetains	: BOOL;
	(* if TRUE, the instance afterwards gets moved into the copy code (online change)*)
	bInCopyCode	: BOOL;
END_VAR
Fatal := TRUE;
END_METHOD

METHOD GetMessage : ERROR_MESSAGE
VAR_INPUT
	showTimestamp : BOOL := FALSE;
	showSource : BOOL := FALSE;
END_VAR
VAR
	stringBuilder : WideStringBuilder;
END_VAR
IF ExceptionCode <> __SYSTEM.ExceptionCode.RTSEXCPT_NOEXCEPTION THEN
	stringBuilder
		.AppendString(SYSTEM_EXCEPTION_PREFIX)
		.Append(ExceptionCode);
			
	IF showTimestamp THEN
		stringBuilder.AppendString(TIME_PREFIX);
		AppendTimestampDescription(stringBuilder);
	END_IF

	stringBuilder.AssignToString(GetMessage);
ELSE
	GetMessage := "";
END_IF
END_METHOD

METHOD INTERNAL SetExceptionCode
VAR_IN_OUT CONSTANT
	exceptionCode : __SYSTEM.ExceptionCode;
END_VAR
THIS^.ExceptionCode := exceptionCode;
THIS^.LocalTimestamp := SystemDateTimeManager.SystemLocalDateTime;
THIS^.UtcTimestamp := SystemDateTimeManager.SystemUtcDateTime;
END_METHOD

END_FUNCTION_BLOCK

// ---- Collections/PointerBased/PointerUniqueSet/PointerUniqueSet.TcPOU
{attribute 'no_explicit_call' := 'do not call this function block directly'} 
// Dynamic set of value pointers
FUNCTION_BLOCK PointerUniqueSet EXTENDS Object IMPLEMENTS IReadOnlyPointerUniqueSet
VAR
	_ClassName : STRING := __POUNAME();
	_Elements : POINTER TO PVOID;
	_ArrayLength : DINT;
	_ElementCount : DINT;
	_DefaultAllocationElemetsCount : BYTE := 10;
	_ElementType : POINTER_TYPE := POINTER_TYPE.BYTE_POINTER;
	_ElementComparer : IComparer;
	_DefaultEnumerator : PointerUniqueSetEnumerator;
END_VAR

METHOD AllocateMemory
VAR_INPUT
	elementsCount : DINT;
END_VAR
VAR
	newElements : POINTER TO PVOID;
END_VAR
newElements := __NEW(PVOID, TO_UDINT(_ArrayLength + elementsCount));

IF _ElementCount > 0 THEN
	Tc2_System.MEMCPY(newElements, _Elements, SIZEOF(POINTER TO BYTE) * TO_UDINT(_ElementCount)); 
END_IF

IF _Elements <> 0 THEN
	__DELETE(_Elements);
END_IF
 
_Elements := newElements;
 
_ArrayLength := _ArrayLength + elementsCount;
END_METHOD

{attribute 'monitoring' := 'call'}
PROPERTY ClassName : STRING
GET
ClassName := _ClassName;
END_GET
END_PROPERTY

METHOD Clear
VAR_INPUT
	deleteElements : BOOL;
END_VAR
VAR
	i : DINT;
	value : PVOID;
END_VAR
IF deleteElements AND_THEN _ElementCount > 0 THEN
	FOR i := 0 TO _ElementCount - 1 DO
		PointerHelper.ReleaseDynamicMemory(_Elements[i], _ElementType);						
	END_FOR	
END_IF

IF _Elements <> 0 THEN
	__DELETE(_Elements);
END_IF

_ElementCount := 0;
_ArrayLength := 0;
END_METHOD

METHOD Contains : BOOL
VAR_INPUT
	element : PVOID;
END_VAR
VAR
	index : DINT; 
END_VAR
Contains := SearchPosition(element, supposedIndex => index);
END_METHOD

{attribute 'OPC.UA.DA.Property' := '1'}
{attribute 'monitoring' := 'call'}
PROPERTY Count : DINT
GET
Count := _ElementCount;
END_GET
END_PROPERTY

{attribute 'OPC.UA.DA.Property' := '1'}
{attribute 'monitoring' := 'call'}
PROPERTY ElementType : POINTER_TYPE
GET
ElementType := _ElementType;
END_GET
END_PROPERTY

METHOD FB_exit : BOOL
VAR_INPUT
	bInCopyCode : BOOL; // if TRUE, the exit method is called for exiting an instance that is copied afterwards (online change).
END_VAR
Clear(FALSE);
END_METHOD

METHOD FB_init : BOOL
VAR_INPUT
	bInitRetains : BOOL; // if TRUE, the retain variables are initialized (warm start / cold start)
	bInCopyCode : BOOL; // if TRUE, the instance afterwards gets moved into the copy code (online change)
	keyType : POINTER_TYPE;
	keyComparer : IComparer;
END_VAR
_DefaultEnumerator.Initialize(THIS^);

_ElementType := keyType;

IF keyComparer = 0 THEN
	_ElementComparer := StandardComparers.GetForType(keyType);
ELSE
	_ElementComparer := keyComparer;
END_IF
END_METHOD

METHOD GetByIndex : PVOID
VAR_INPUT
	index : DINT;
END_VAR
IF index >= 0 AND index < _ElementCount THEN
	GetByIndex := _Elements[index];
END_IF
END_METHOD

METHOD GetDefaultEnumerator : IEnumerator
GetDefaultEnumerator := _DefaultEnumerator;
END_METHOD

METHOD Remove : BOOL
VAR_INPUT
	element : PVOID;
	delete : BOOL;
END_VAR
VAR
	index : DINT;
END_VAR
IF SearchPosition(element, supposedIndex => index) THEN
	RemoveAt(index, delete);
	Remove := TRUE;
END_IF
END_METHOD

METHOD RemoveAt : BOOL
VAR_INPUT
	index : DINT;
	delete : BOOL;
END_VAR
VAR
	i : DINT;
END_VAR
IF index < _ElementCount THEN
	IF delete THEN
		PointerHelper.ReleaseDynamicMemory(_Elements[index], _ElementType);			
	END_IF
	
	IF index + 2 <= _ElementCount THEN
		FOR	i := index TO _ElementCount - 2 DO
			_Elements[i] := _Elements[i + 1];
		END_FOR
	END_IF	
		
	_Elements[_ElementCount - 1] := 0;
	_ElementCount := _ElementCount - 1;
	
	RemoveAt := TRUE;
END_IF
END_METHOD

METHOD PROTECTED SearchPosition : BOOL
VAR_INPUT
	element : PVOID;
END_VAR
VAR_OUTPUT
	supposedIndex : DINT; 
END_VAR
VAR
	currentElement : PVOID;
	lastIndex : DINT;
	minIndex : DINT;
	maxIndex : DINT;
END_VAR
IF _ElementCount = 0 THEN
	RETURN;
END_IF

lastIndex := _ElementCount - 1;
maxIndex := lastIndex;
supposedIndex := maxIndex / 2;

WHILE minIndex <= maxIndex DO
	currentElement := _Elements[supposedIndex];
	
	CASE _ElementComparer.Compare(currentElement, element) OF
		// assumed key equals to seached 
		COMPARISION_RESULT.EQUALS:
			SearchPosition := TRUE;
			RETURN;

		// assumed key less than searched, move range to right
		COMPARISION_RESULT.LEFT_LESS_RIGHT:
			minIndex := supposedIndex + 1;
			
		// assumed key greater than searched, move range to left	
		COMPARISION_RESULT.LEFT_GREATER_RIGHT:
			maxIndex := supposedIndex - 1;
	END_CASE
	
	supposedIndex := minIndex + (maxIndex - minIndex) / 2;
END_WHILE
END_METHOD

METHOD Set : DINT
VAR_INPUT
	element : PVOID;
	deleteReplacedElement : BOOL;
END_VAR
VAR
	index, i : DINT;
END_VAR
// if equal key found then we need to replace it
IF SearchPosition(element, supposedIndex => index) THEN	
	// old and new keys show to diffirent address, then we need to replace existing key 
	IF _Elements[index] <> element THEN
		IF deleteReplacedElement THEN
			PointerHelper.ReleaseDynamicMemory(_Elements[index], _ElementType);
		END_IF
		
		_Elements[index] := element;
	END_IF
// if equal key not found than we need to insert it
ELSE
	IF _ElementCount >= _ArrayLength THEN
		AllocateMemory(_DefaultAllocationElemetsCount);
	END_IF
	
	i := _ElementCount;	
	_ElementCount := _ElementCount + 1;
		
	WHILE i > index DO
		_Elements[i] := _Elements[i - 1];
		
		i := i - 1;
	END_WHILE
	
	_Elements[index] := element;
END_IF

Set := index;
END_METHOD

END_FUNCTION_BLOCK

// ---- Collections/PointerBased/PointerUniqueSet/PointerUniqueSetEnumerator.TcPOU
{attribute 'no_explicit_call' := 'do not call this function block directly'} 
{attribute 'enable_dynamic_creation'}
FUNCTION_BLOCK PointerUniqueSetEnumerator EXTENDS Enumerator
VAR
	_ClassName : STRING := __POUNAME();
	_HashSet : IReadOnlyPointerUniqueSet;
	_Current : PVOID;
END_VAR

{attribute 'monitoring' := 'call'}
PROPERTY ClassName : STRING
GET
ClassName := _ClassName;
END_GET
END_PROPERTY

{attribute 'OPC.UA.DA.Property' := '1'}
{attribute 'monitoring' := 'call'}
PROPERTY Current : PVOID
GET
Current := ADR(_Current);
END_GET
END_PROPERTY

METHOD INTERNAL Initialize 
VAR_INPUT
	hashSet : IReadOnlyPointerUniqueSet;
END_VAR
_HashSet := hashSet;
END_METHOD

{attribute "object_name" := "MoveNext"}
METHOD MoveNext : BOOL
_CurrentIndex := _CurrentIndex + 1;

IF _CurrentIndex >= _HashSet.Count THEN
	_Current := 0;
	_CurrentIndex := _HashSet.Count;
ELSE
	_Current := _HashSet.GetByIndex(_CurrentIndex);	
	MoveNext := TRUE;
END_IF
END_METHOD

{attribute "object_name" := "Reset"}
METHOD Reset
SUPER^.Reset();

_Current := 0;
END_METHOD

END_FUNCTION_BLOCK

// ---- Collections/PointerBased/PointerList/PointerList.TcPOU
{attribute 'no_explicit_call' := 'do not call this function block directly'} 
// Dynamic list of value pointers
FUNCTION_BLOCK PointerList EXTENDS Object IMPLEMENTS IReadOnlyPointerList
VAR_INPUT
	DefaultAllocationElemetsCount : BYTE := 10;	
END_VAR
VAR
	_ClassName : STRING := __POUNAME();
	_Array : POINTER TO PVOID;
	_ArrayLength : DINT;
	_ElementCount : DINT;
	_ElementType : POINTER_TYPE := POINTER_TYPE.BYTE_POINTER;
	_DefaultComparer : IComparer;
	_DefaultEnumerator : PointerListEnumerator;
END_VAR

METHOD AllocateMemory
VAR_INPUT
	elementsCount : DINT;
END_VAR
VAR
	
	newMemory : POINTER TO PVOID;
END_VAR
newMemory := __NEW(PVOID, TO_UDINT(_ArrayLength + elementsCount));

IF _ElementCount > 0 THEN
	Tc2_System.MEMCPY(newMemory, _Array, TO_UDINT(SIZEOF(POINTER TO BYTE) * _ElementCount));
END_IF
 
IF _Array <> 0 THEN
	__DELETE(_Array);
END_IF

_ArrayLength := _ArrayLength + elementsCount;

_Array := newMemory;
END_METHOD

METHOD Append : DINT
VAR_INPUT
	element : PVOID;
END_VAR
Append := _ElementCount;

Insert(element, Append);
END_METHOD

{attribute 'monitoring' := 'call'}
PROPERTY ClassName : STRING
GET
ClassName := _ClassName;
END_GET
END_PROPERTY

METHOD Clear
VAR_INPUT
	delete : BOOL;
END_VAR
VAR
	i : DINT;
END_VAR
IF delete AND_THEN _ElementCount > 0 THEN
	FOR i := _ElementCount - 1 TO 0 BY -1 DO 
		PointerHelper.ReleaseDynamicMemory(_Array[i], _ElementType);						
	END_FOR	
END_IF

_ElementCount := 0;
_ArrayLength := 0;

IF _Array <> 0 THEN
	__DELETE(_Array);	
END_IF
END_METHOD

{attribute 'OPC.UA.DA.Property' := '1'}
{attribute 'monitoring' := 'call'}
PROPERTY Count : DINT
GET
Count := _ElementCount;
END_GET
END_PROPERTY

{attribute 'OPC.UA.DA.Property' := '1'}
{attribute 'monitoring' := 'call'}
PROPERTY ElementType : POINTER_TYPE
GET
ElementType := _ElementType;
END_GET
END_PROPERTY

METHOD FB_exit : BOOL
VAR_INPUT
	bInCopyCode : BOOL; // if TRUE, the exit method is called for exiting an instance that is copied afterwards (online change).
END_VAR
Clear(FALSE);
END_METHOD

METHOD FB_init : BOOL
VAR_INPUT
	bInitRetains : BOOL; // if TRUE, the retain variables are initialized (warm start / cold start)
	bInCopyCode : BOOL; // if TRUE, the instance afterwards gets moved into the copy code (online change)
	elementType : POINTER_TYPE;
END_VAR
_DefaultEnumerator.Initialize(THIS^);

_ElementType := elementType;

_DefaultComparer := StandardComparers.GetForType(elementType);
END_METHOD

METHOD Find : BOOL
VAR_INPUT
	pattern : PVOID;
	comparer : IComparer;
	skip : DINT;
END_VAR
VAR_OUTPUT
	element : PVOID;
	index : DINT;
END_VAR
VAR
	i : DINT;
	skiped : DINT := 0;
END_VAR
element := 0;
index := 0;
	
IF skip >= _ElementCount THEN
	RETURN;
END_IF

IF comparer = 0 THEN
	comparer := StandardComparers.GetForType(_ElementType);
END_IF

IF _ElementCount > 0 THEN
	FOR i := 0 TO _ElementCount - 1 DO
		IF comparer.Compare(_Array[i], pattern) = COMPARISION_RESULT.EQUALS THEN
			IF skip = skiped THEN
				element := _Array[i];
				index := i;
				Find := TRUE;
				RETURN;
			ELSE
				skiped := skiped + 1;
			END_IF
		END_IF
	END_FOR
END_IF
END_METHOD

METHOD Get : PVOID
VAR_INPUT
	index : DINT;
END_VAR
IF index >= 0 AND index < _ElementCount THEN
	Get := _Array[index];
ELSE
	Get := 0;
END_IF
END_METHOD

METHOD GetDefaultEnumerator : IEnumerator
GetDefaultEnumerator := _DefaultEnumerator;
END_METHOD

METHOD Insert
VAR_INPUT
	element : PVOID;
	index : DINT;
END_VAR
VAR
	i : DINT;
END_VAR
IF index > Count THEN
	index := _ElementCount;
END_IF

IF _ElementCount >= _ArrayLength THEN
	AllocateMemory(DefaultAllocationElemetsCount);
END_IF

_ElementCount := _ElementCount + 1;

i := _ElementCount - 1;

WHILE i > index DO
	_Array[i] := _Array[i - 1];
	
	i := i - 1;
END_WHILE

_Array[i] := element;
END_METHOD

METHOD Remove : BOOL
VAR_INPUT
	element : PVOID;
	delete : BOOL;
END_VAR
VAR
	i : DINT;
END_VAR
IF _ElementCount > 0 THEN
	FOR i := 0 TO _ElementCount - 1 DO
		IF _Array[i] = element THEN
			RemoveAt(i, delete);
			Remove := TRUE;
			RETURN;
		END_IF
	END_FOR
END_IF
END_METHOD

METHOD RemoveAt : BOOL
VAR_INPUT
	index : DINT;
	delete : BOOL;
END_VAR
VAR
	i : DINT;
END_VAR
IF index < _ElementCount THEN
	IF delete THEN
		PointerHelper.ReleaseDynamicMemory(_Array[index], _ElementType);			
	END_IF	

	IF index + 2 <= _ElementCount THEN
		FOR	i := index TO _ElementCount - 2 DO
			_Array[i] := _Array[i + 1];
		END_FOR			
	END_IF
		
	_Array[_ElementCount - 1] := 0;
	_ElementCount := _ElementCount - 1;
	
	RemoveAt := TRUE;
END_IF
END_METHOD

METHOD Set : BOOL
VAR_INPUT
	element : PVOID;
	index : DINT;
	deleteReplaced : BOOL;
END_VAR
IF index >= 0 AND_THEN index < _ElementCount THEN
	IF _Array[index] <> element THEN
		IF deleteReplaced THEN
			PointerHelper.ReleaseDynamicMemory(_Array[index], _ElementType);
		END_IF
	
		_Array[index] := element;
	END_IF
	
	Set := TRUE;
ELSE
	Set := FALSE;
END_IF
END_METHOD

METHOD Sort
VAR_INPUT
	comparer : IComparer;
	direction : SORTING_DIRECTION;
END_VAR
VAR
	//exceptionFactory : ExceptionFactory(__POUNAME(), ClassName, CurrentNamespace.Name);
	replaced : BOOL;
	i : DINT;
	comparisionResult : COMPARISION_RESULT;
END_VAR
IF comparer = 0 THEN
	IF _DefaultComparer = 0 THEN
		//exceptionFactory.ThrowException(__POSITION(), WStringHelper.Concat2("Can't find comparer for POINTER TO ", TO_WSTRING(_ElementType)));
	ELSE
		comparer := _DefaultComparer;
	END_IF
END_IF

REPEAT
	replaced := FALSE;
	
	IF _ElementCount > 1 THEN
		FOR i := 0 TO _ElementCount - 2 DO
			comparisionResult := comparer.Compare(_Array[i], _Array[i + 1]);
			
			IF direction = SORTING_DIRECTION.ASCENDING THEN
				IF comparisionResult = COMPARISION_RESULT.LEFT_GREATER_RIGHT THEN
					Swap(i, i + 1);
					replaced := TRUE;
				END_IF
			ELSE
				IF comparisionResult = COMPARISION_RESULT.LEFT_LESS_RIGHT THEN
					Swap(i, i + 1);
					replaced := TRUE;
				END_IF			
			END_IF
		END_FOR		
	END_IF
UNTIL
	NOT replaced
END_REPEAT
END_METHOD

METHOD Swap : BOOL
VAR_INPUT
	index1 : DINT;
	index2 : DINT;
END_VAR
VAR
	tmp : PVOID;
END_VAR
IF index1 = index2 OR_ELSE index1 < 0 OR_ELSE index1 >= _ElementCount OR_ELSE index2 < 0 OR_ELSE index2 >= _ElementCount THEN
	RETURN;
END_IF

tmp := _Array[index1];
_Array[index1] := _Array[index2];
_Array[index2] := tmp;

Swap := TRUE;
END_METHOD

END_FUNCTION_BLOCK

// ---- Collections/PointerBased/PointerList/PointerListEnumerator.TcPOU
{attribute 'no_explicit_call' := 'do not call this function block directly'} 
{attribute 'enable_dynamic_creation'}
FUNCTION_BLOCK PointerListEnumerator EXTENDS Enumerator
VAR
	_ClassName : STRING := __POUNAME();
	_List : IReadOnlyPointerList;
	_Current : PVOID;
END_VAR

{attribute 'monitoring' := 'call'}
PROPERTY ClassName : STRING
GET
ClassName := _ClassName;
END_GET
END_PROPERTY

PROPERTY Current : PVOID
GET
Current := _Current;
END_GET
END_PROPERTY

METHOD INTERNAL Initialize
VAR_INPUT
	list : IReadOnlyPointerList;
END_VAR
_List := list;
END_METHOD

{attribute "object_name" := "MoveNext"}
METHOD MoveNext : BOOL
_CurrentIndex := _CurrentIndex + 1;

IF _CurrentIndex >= _List.Count THEN
	_Current := 0;	
	_CurrentIndex := _List.Count;
ELSE
	_Current := _List.Get(_CurrentIndex);	
	MoveNext := TRUE;
END_IF
END_METHOD

{attribute "object_name" := "Reset"}
METHOD Reset
SUPER^.Reset();

_Current := 0;
END_METHOD

END_FUNCTION_BLOCK

// ---- Collections/ValueBased/ByteList/ByteList.TcPOU
{attribute 'no_explicit_call' := 'do not call this function block directly'} 
{attribute 'enable_dynamic_creation'}
// Collection of bytes of dynamic size
FUNCTION_BLOCK ByteList EXTENDS Object IMPLEMENTS IByteList
VAR_OUTPUT
	DataAddress : POINTER TO BYTE;
END_VAR
VAR
	_ClassName : STRING := __POUNAME();
	_MemorySize : DINT;
	_BytesCount : DINT;
	_DefaultEnumerator : ByteListEnumerator;
END_VAR

{attribute 'OPC.UA.DA.Property' := '1'}
{attribute 'monitoring' := 'call'}
PROPERTY Address : POINTER TO BYTE
GET
Address := DataAddress;
END_GET
END_PROPERTY

METHOD Append
VAR_INPUT
	value : BYTE;
END_VAR
VAR
	newMemory : POINTER TO BYTE;
END_VAR
// if existing memory is not enough
IF _BytesCount >= _MemorySize THEN
	// calculate new memory size
	_MemorySize := _BytesCount + 1;
	
	// allocate new memory
	newMemory := __NEW(BYTE, TO_UDINT(_MemorySize));
	
	// copy existing bytes to new memory if needed
	IF _BytesCount > 0 THEN
		Tc2_System.MEMCPY(newMemory, DataAddress, TO_UDINT(_BytesCount));		
	END_IF
	
	// release old memory
	IF DataAddress <> 0 THEN
		__DELETE(DataAddress);		
	END_IF
	
	// save new memory reference
	DataAddress := newMemory;
END_IF

// append new bytes
Tc2_System.MEMCPY(DataAddress + TO_DWORD(_BytesCount), ADR(value), 1);

// set new bytes count
_BytesCount := _BytesCount + 1;
END_METHOD

{attribute 'monitoring' := 'call'}
PROPERTY ClassName : STRING
GET
ClassName := _ClassName;
END_GET
END_PROPERTY

METHOD Clear
VAR_INPUT
	releaseMemory : BOOL := FALSE;
END_VAR
IF releaseMemory AND_THEN _MemorySize > 0 THEN
	__DELETE(DataAddress);
	_MemorySize := 0;
END_IF

_BytesCount := 0;
END_METHOD

{attribute 'OPC.UA.DA.Property' := '1'}
{attribute 'monitoring' := 'call'}
PROPERTY Count : DINT
GET
Count := _BytesCount;
END_GET
END_PROPERTY

METHOD FB_exit : BOOL
VAR_INPUT
	bInCopyCode : BOOL; // if TRUE, the exit method is called for exiting an instance that is copied afterwards (online change).
END_VAR
IF DataAddress <> 0 THEN
	__DELETE(DataAddress);
END_IF
END_METHOD

METHOD FB_init : BOOL
VAR_INPUT
	(* if TRUE, the retain variables are initialized (warm start / cold start)*)
	bInitRetains	: BOOL;
	(* if TRUE, the instance afterwards gets moved into the copy code (online change)*)
	bInCopyCode	: BOOL;
END_VAR
_DefaultEnumerator.Initialize(THIS^);
END_METHOD

METHOD Find : BOOL
VAR_INPUT
	value : BYTE;
END_VAR
VAR_OUTPUT
	index : DINT;
END_VAR
VAR
	i : DINT;	
END_VAR
IF _BytesCount > 0 THEN
	FOR i := 0 TO _BytesCount - 1 DO
		IF DataAddress[i] = value THEN
			index := i;
			Find := TRUE;
			RETURN;
		END_IF 	
	END_FOR
END_IF
END_METHOD

METHOD Get : BYTE
VAR_INPUT
	index : DINT;
END_VAR
VAR
	exception : StandardException;
END_VAR
IF DataAddress = 0 THEN
	exception.Throw(CurrentNamespace.Name, ClassName, __POUNAME(), __POSITION(), "Dynamic byte array is empty");
END_IF

IF index < 0 THEN
	exception.Throw(CurrentNamespace.Name, ClassName, __POUNAME(), __POSITION(), "Index is less then zero");
END_IF

IF index >= _BytesCount THEN
	exception.Throw(CurrentNamespace.Name, ClassName, __POUNAME(), __POSITION(), "Index is too large");
END_IF

Get := DataAddress[index];
END_METHOD

METHOD GetDefaultEnumerator : IEnumerator
GetDefaultEnumerator := _DefaultEnumerator;
END_METHOD

METHOD LoadFromAddress
VAR_INPUT
	startIndex : DINT;
	sourceDataAddress : POINTER TO BYTE;
	sourceDataSize : DINT;
END_VAR
VAR
	exception : StandardException;
	newMemory : POINTER TO BYTE;
END_VAR
IF startIndex < 0 THEN
	exception.Throw(CurrentNamespace.Name, ClassName, __POUNAME(), __POSITION(), "Start index is less then zero");
END_IF

IF startIndex > _BytesCount THEN
	exception.Throw(CurrentNamespace.Name, ClassName, __POUNAME(), __POSITION(), "Start index is too large");
END_IF

IF sourceDataSize < 0 THEN
	exception.Throw(CurrentNamespace.Name, ClassName, __POUNAME(), __POSITION(), "Source bytes count is less then zero");
END_IF

IF sourceDataAddress = 0 OR_ELSE sourceDataSize = 0 THEN
	RETURN;
END_IF

IF startIndex + sourceDataSize > _MemorySize THEN
	// calculate new memory size
	_MemorySize := startIndex + sourceDataSize;
	
	// allocate new memory
	newMemory := __NEW(BYTE, TO_UDINT(_MemorySize));
	
	// copy existing bytes to new memory if needed
	IF startIndex > 0 THEN
		MEMCPY(newMemory, DataAddress, TO_UDINT(startIndex));		
	END_IF
	
	// append new bytes
	MEMCPY(newMemory + TO_DWORD(startIndex), sourceDataAddress, TO_UDINT(sourceDataSize));
	
	// set new bytes count
	_BytesCount := _MemorySize;
	
	// release old memory
	IF DataAddress <> 0 THEN
		__DELETE(DataAddress);		
	END_IF
	
	// save new memory reference
	DataAddress := newMemory;
ELSE
	// append new bytes
	MEMCPY(DataAddress + TO_DWORD(startIndex), sourceDataAddress, TO_UDINT(sourceDataSize));
	
	// set new bytes count
	_BytesCount := startIndex + sourceDataSize;	
END_IF
END_METHOD

METHOD LoadFromVariable
VAR_INPUT
	startIndex : DINT;
	sourceVariable : ANY;
END_VAR
VAR
	exception : StandardException;
	newMemory : POINTER TO BYTE;
END_VAR
IF startIndex < 0 THEN
	exception.Throw(CurrentNamespace.Name, ClassName, __POUNAME(), __POSITION(), "Start index is less then zero");
END_IF

IF startIndex > _BytesCount THEN
	exception.Throw(CurrentNamespace.Name, ClassName, __POUNAME(), __POSITION(), "Start index is too large");
END_IF

IF sourceVariable.pValue = 0 OR_ELSE sourceVariable.diSize = 0 THEN
	RETURN;
END_IF

LoadFromAddress(startIndex, sourceVariable.pValue, sourceVariable.diSize);
END_METHOD

METHOD Remove
VAR_INPUT
	value : BYTE;
	freeUnusedMemory : BOOL := FALSE;
END_VAR
VAR
	index : DINT;
	exception : StandardException;
END_VAR
IF DataAddress = 0 THEN
	exception.Throw(CurrentNamespace.Name, ClassName, __POUNAME(), __POSITION(), "Dynamic byte array is empty");
END_IF

IF count < 0 THEN
	exception.Throw(CurrentNamespace.Name, ClassName, __POUNAME(), __POSITION(), "Count is less then zero");
END_IF

IF index + count > _BytesCount THEN
	exception.Throw(CurrentNamespace.Name, ClassName, __POUNAME(), __POSITION(), "Index + count are outside the array bounds");
END_IF

IF Find(value, index => index) THEN
	RemoveAt(index, 1, freeUnusedMemory);
END_IF
END_METHOD

METHOD RemoveAt
VAR_INPUT
	index : DINT;
	count : DINT := 1;
	freeUnusedMemory : BOOL := FALSE;
END_VAR
VAR
	exception : StandardException;
	newMemory : POINTER TO BYTE;
END_VAR
IF DataAddress = 0 THEN
	exception.Throw(CurrentNamespace.Name, ClassName, __POUNAME(), __POSITION(), "Dynamic byte array is empty");
END_IF

IF index < 0 THEN
	exception.Throw(CurrentNamespace.Name, ClassName, __POUNAME(), __POSITION(), "Index is less then zero");
END_IF

IF count < 0 THEN
	exception.Throw(CurrentNamespace.Name, ClassName, __POUNAME(), __POSITION(), "Count is less then zero");
END_IF

IF index + count > _BytesCount THEN
	exception.Throw(CurrentNamespace.Name, ClassName, __POUNAME(), __POSITION(), "Index + count are outside the array bounds");
END_IF

IF freeUnusedMemory THEN
	// calculate new memory size
	_MemorySize := _BytesCount - count;
	
	// allocate new memory
	newMemory := __NEW(BYTE, TO_UDINT(_MemorySize)); 
	
	// copy leading bytes if needed
	IF index <> 0 THEN
		Tc2_System.MEMCPY(newMemory, DataAddress, TO_UDINT(index));
	END_IF
	
	// copy trailing bytes
	Tc2_System.MEMCPY(newMemory + TO_DWORD(index), DataAddress + TO_DWORD(index + count), TO_UDINT(_BytesCount - index - count));
	
	// release old buffer
	__DELETE(DataAddress);
	
	// save new buffer
	DataAddress := newMemory;

	// set bytes count
	_BytesCount := _MemorySize;	
ELSE
	// copy trailing bytes
	Tc2_System.MEMCPY(DataAddress + TO_DWORD(index), DataAddress + TO_DWORD(index + count), TO_UDINT(_BytesCount - index - count));

	// set bytes count
	_BytesCount := _BytesCount - count;
END_IF
END_METHOD

METHOD Resize
VAR_INPUT
	newBytesCount : DINT; // in bytes
END_VAR
VAR
	exception : StandardException;
	newMemory : POINTER TO BYTE;
END_VAR
IF newBytesCount < 0 THEN
	exception.Throw(CurrentNamespace.Name, ClassName, __POUNAME(), __POSITION(), "New bytes count is less then zero");
END_IF

// if existing memory is not enough
IF newBytesCount > _MemorySize THEN
	// calculate new memory size
	_MemorySize := newBytesCount;
	
	// allocate new memory
	newMemory := __NEW(BYTE, TO_UDINT(_MemorySize));
	
	// copy existing bytes to new memory if needed
	IF _BytesCount > 0 THEN
		Tc2_System.MEMCPY(newMemory, DataAddress, TO_UDINT(_BytesCount));		
	END_IF
	
	// release old memory
	IF DataAddress <> 0 THEN
		__DELETE(DataAddress);		
	END_IF
	
	// save new memory reference
	DataAddress := newMemory;
END_IF

// set new bytes count
_BytesCount := newBytesCount;
END_METHOD

METHOD Set
VAR_INPUT
	index : DINT;
	value : BYTE;
END_VAR
VAR
	exception : StandardException;
END_VAR
IF DataAddress = 0 THEN
	exception.Throw(CurrentNamespace.Name, ClassName, __POUNAME(), __POSITION(), "Dynamic byte array is empty");
END_IF

IF index < 0 THEN
	exception.Throw(CurrentNamespace.Name, ClassName, __POUNAME(), __POSITION(), "Index is less then zero");
END_IF

IF index >= _BytesCount THEN
	exception.Throw(CurrentNamespace.Name, ClassName, __POUNAME(), __POSITION(), "Index is too large");
END_IF

DataAddress[index] := value;
END_METHOD

END_FUNCTION_BLOCK

// ---- Collections/ValueBased/ByteList/ByteListEnumerator.TcPOU
{attribute 'no_explicit_call' := 'do not call this function block directly'} 
{attribute 'enable_dynamic_creation'}
FUNCTION_BLOCK ByteListEnumerator EXTENDS Enumerator
VAR
	_ClassName : STRING := __POUNAME();
	_List : IReadOnlyByteList;
	_Current : POINTER TO BYTE;
END_VAR

{attribute 'monitoring' := 'call'}
PROPERTY ClassName : STRING
GET
ClassName := _ClassName;
END_GET
END_PROPERTY

{attribute 'OPC.UA.DA.Property' := '1'}
{attribute 'monitoring' := 'call'}
PROPERTY Current : PVOID
GET
Current := _Current;
END_GET
END_PROPERTY

METHOD INTERNAL Initialize
VAR_INPUT
	list : IReadOnlyByteList;
END_VAR
_List := list;
END_METHOD

{attribute "object_name" := "MoveNext"}
METHOD MoveNext : BOOL
_CurrentIndex := _CurrentIndex + 1;	

IF _CurrentIndex >= _List.Count THEN
	_Current := 0;
	_CurrentIndex := _List.Count;
ELSE
	_Current := _List.Get(_CurrentIndex);	
	MoveNext := TRUE;
END_IF
END_METHOD

{attribute "object_name" := "Reset"}
METHOD Reset
SUPER^.Reset();

_Current := 0;
END_METHOD

END_FUNCTION_BLOCK

// ---- Exceptions/General/Standard/StandardException.TcPOU
{attribute 'enable_dynamic_creation'}	
{attribute 'no_explicit_call' := 'do not call this function block directly'} 
FUNCTION_BLOCK StandardException EXTENDS GeneralException
VAR
	_ClassName : STRING := __POUNAME();
END_VAR

{attribute 'monitoring' := 'call'}
PROPERTY ClassName : STRING
GET
ClassName := _ClassName;
END_GET
END_PROPERTY

METHOD Clone : IObject
VAR
	exceptionClone : POINTER TO StandardException;
END_VAR
exceptionClone := __NEW(StandardException);

Clone := InternalClone(exceptionClone);
END_METHOD

METHOD Throw
VAR_INPUT
	sourceNamespaceName : STRING;
	sourceClassName : STRING;
	sourceMethodName : STRING;
	sourcePosition : STRING;
	message : ERROR_MESSAGE;
	errorCode : UDINT := 0;
	fatal : BOOL := FALSE;
	innerException : REFERENCE TO Exception REF= 0;
END_VAR
InternalThrow(sourceNamespaceName, sourceClassName, sourceMethodName, sourcePosition, message, errorCode, fatal, innerException);
END_METHOD

END_FUNCTION_BLOCK

// ---- Comparing/StandardComparers/LDateAndTimeComparer.TcPOU
FUNCTION_BLOCK LDateAndTimeComparer EXTENDS Object IMPLEMENTS IComparer
VAR
	_ClassName : STRING := __POUNAME();
END_VAR

{attribute 'monitoring' := 'call'}
PROPERTY ClassName : STRING
GET
ClassName := _ClassName;
END_GET
END_PROPERTY

{attribute "object_name" := "Compare"}
METHOD Compare : COMPARISION_RESULT
VAR_INPUT
	left : PVOID;
	right : PVOID;
END_VAR
VAR
	leftPointer : POINTER TO LDATE_AND_TIME; 
	rightPointer : POINTER TO LDATE_AND_TIME; 
END_VAR
IF left = 0 AND right = 0 THEN
	Compare := COMPARISION_RESULT.EQUALS;
	RETURN;
END_IF

IF left = 0 THEN
	Compare := COMPARISION_RESULT.LEFT_LESS_RIGHT;
	RETURN;	
END_IF

IF right = 0 THEN
	Compare := COMPARISION_RESULT.LEFT_GREATER_RIGHT;
	RETURN;	
END_IF

leftPointer := left;
rightPointer := right;

IF leftPointer^ < rightPointer^ THEN
	Compare := COMPARISION_RESULT.LEFT_LESS_RIGHT;
ELSIF leftPointer^ > rightPointer^ THEN
	Compare := COMPARISION_RESULT.LEFT_GREATER_RIGHT;
ELSE
	Compare := COMPARISION_RESULT.EQUALS;	
END_IF
END_METHOD

END_FUNCTION_BLOCK

// ---- Exceptions/Aggregate/AggregateException.TcPOU
{attribute 'enable_dynamic_creation'}	
{attribute 'no_explicit_call' := 'do not call this function block directly'} 
FUNCTION_BLOCK AggregateException EXTENDS Exception
VAR
	_ClassName : STRING := __POUNAME();
	_InnerExceptions : POINTER TO IException;
	_InnerExceptionCount : UINT;
END_VAR
VAR CONSTANT
	EXCEPTION_NUMBER_DELIMITER : WSTRING(1) := ".";
	AGGREGATE_EXCEPTION_SUFFIX : WSTRING(25) := " aggregated exceptions";
END_VAR

METHOD AddInnerException
VAR_IN_OUT CONSTANT
	innerException : IException; // will be cloned
END_VAR
VAR
	innerExceptionClone : IException;
	newInnerExceptions : POINTER TO IException;
END_VAR
__QUERYINTERFACE(innerException.Clone(), innerExceptionClone); 

newInnerExceptions := __NEW(POINTER TO IException, (_InnerExceptionCount + 1));
	
Tc2_System.MEMCPY(newInnerExceptions, _InnerExceptions, TO_UDINT(SIZEOF(POINTER TO IException) * _InnerExceptionCount));

newInnerExceptions[_InnerExceptionCount] := innerExceptionClone; 

_InnerExceptionCount := _InnerExceptionCount + 1;
END_METHOD

{attribute 'monitoring' := 'call'}
PROPERTY ClassName : STRING
GET
ClassName := _ClassName;
END_GET
END_PROPERTY

METHOD Clone : IObject
VAR
	exceptionClone : POINTER TO AggregateException;
	i : DINT;
	innerException : POINTER TO Exception;
END_VAR
exceptionClone := __NEW(AggregateException);

exceptionClone^.Fatal := Fatal;
exceptionClone^.SourceNamespaceName := SourceNamespaceName;
exceptionClone^.SourceClassName := SourceClassName;
exceptionClone^.SourceMethodName := SourceMethodName;
exceptionClone^.SourcePosition := SourcePosition;
exceptionClone^.LocalTimestamp := LocalTimestamp;	
exceptionClone^.UtcTimestamp := UtcTimestamp;	

FOR i := 0 TO _InnerExceptionCount - 1 DO
	exceptionClone^.AddInnerException(_InnerExceptions[i]);
END_FOR

Clone := exceptionClone^;
END_METHOD

{attribute 'monitoring' := 'call'}
PROPERTY Empty : BOOL
GET
Empty := _InnerExceptionCount = 0;
END_GET
END_PROPERTY

METHOD FB_exit : BOOL
VAR_INPUT
	(* if TRUE, the exit method is called for exiting an instance that is copied afterwards (online change).*)
	bInCopyCode	: BOOL;
END_VAR
VAR
	i : DINT;
END_VAR
FOR i := 0 TO _InnerExceptionCount - 1 DO
	_InnerExceptions[i].Dispose();
END_FOR
END_METHOD

METHOD GetMessage : ERROR_MESSAGE
VAR_INPUT
	showTimestamp : BOOL := FALSE;
	showSource : BOOL := FALSE;
END_VAR
VAR
	stringBuilder : WideStringBuilder;
	
	i : DINT;
	innerExceptionMessage : ERROR_MESSAGE;
END_VAR
stringBuilder
	.Append(_InnerExceptionCount)
	.AppendString(AGGREGATE_EXCEPTION_SUFFIX);

IF showTimestamp THEN
	stringBuilder.AppendString(TIME_PREFIX);
	AppendTimestampDescription(stringBuilder);
END_IF

IF showSource THEN
	stringBuilder.AppendString(SOURCE_PREFIX);
	AppendSourceDescription(stringBuilder);
END_IF

FOR i := 0 TO _InnerExceptionCount - 1 DO
	innerExceptionMessage := _InnerExceptions[i].GetMessage(showTimestamp, showSource);
	
	stringBuilder
		.AppendString(WideStringHelper.NewLine)
		.Append(i)
		.AppendString(EXCEPTION_NUMBER_DELIMITER)	
		.Append(innerExceptionMessage);
END_FOR		

stringBuilder.AssignToString(GetMessage);
END_METHOD

PROPERTY InnerExceptionCount : UINT
GET
InnerExceptionCount := _InnerExceptionCount;
END_GET
END_PROPERTY

PROPERTY InnerExceptions : POINTER TO IException
GET
InnerExceptions := _InnerExceptions;
END_GET
END_PROPERTY

METHOD Throw
VAR_INPUT
	sourceNamespaceName : STRING;
	sourceClassName : STRING;
	sourceMethodName : STRING;
	sourcePosition : STRING;
END_VAR
VAR
	i : DINT;
END_VAR
THIS^.SourceNamespaceName := sourceNamespaceName;	
THIS^.SourceClassName := sourceClassName;
THIS^.SourceMethodName := SEL(Tc2_Standard.FIND(sourceMethodName, sourceClassName) <> 1, Tc2_Standard.DELETE(sourceMethodName, Tc2_Standard.LEN(sourceClassName) + 1, 1), sourceMethodName); 
THIS^.SourcePosition := sourcePosition;
THIS^.Fatal := FALSE;
THIS^.LocalTimestamp := SystemDateTimeManager.SystemLocalDateTime;
THIS^.UtcTimestamp := SystemDateTimeManager.SystemUtcDateTime;

FOR i := 0 TO _InnerExceptionCount - 1 DO
	IF _InnerExceptions[i].Fatal THEN
		THIS^.Fatal := TRUE;
		EXIT;
	END_IF
END_FOR

ExceptionManager.Throw(THIS^);
END_METHOD

END_FUNCTION_BLOCK

// ---- Exceptions/General/NotImplemented/NotImplementedException.TcPOU
{attribute 'enable_dynamic_creation'}	
{attribute 'no_explicit_call' := 'do not call this function block directly'} 
FUNCTION_BLOCK NotImplementedException EXTENDS GeneralException
VAR
	_ClassName : STRING := __POUNAME();
END_VAR

{attribute 'monitoring' := 'call'}
PROPERTY ClassName : STRING
GET
ClassName := _ClassName;
END_GET
END_PROPERTY

METHOD Clone : IObject
VAR
	exceptionClone : POINTER TO NotImplementedException;
END_VAR
exceptionClone := __NEW(NotImplementedException);

Clone := InternalClone(exceptionClone);
END_METHOD

METHOD Throw
VAR_INPUT
	sourceNamespaceName : STRING;
	sourceClassName : STRING;
	sourceMethodName : STRING;
	sourcePosition : STRING;
	fatal : BOOL := FALSE;
END_VAR
VAR
	stringBuilder : WideStringBuilder;
	message : ERROR_MESSAGE;
	nullInnerException : REFERENCE TO Exception REF= 0;
END_VAR
stringBuilder.AppendString("Program organization unit '");

AppendProgramOrganizationUnitFullName(stringBuilder);

stringBuilder
	.AppendString(" ' is not implemented")
	.AssignToString(message);

InternalThrow(sourceNamespaceName, sourceClassName, sourceMethodName, sourcePosition, message, errorCode, fatal, nullInnerException);
END_METHOD

END_FUNCTION_BLOCK

// ---- Helpers/MathHelper.TcPOU
PROGRAM MathHelper
VAR
	_Random : DRAND;
END_VAR

METHOD ConvertDegreesToRadians : LREAL
VAR_INPUT
	degrees : LREAL;
END_VAR
ConvertDegreesToRadians := degrees * PI / 180;
END_METHOD

METHOD ConvertRadiansToDegrees : LREAL
VAR_INPUT
	radiand : LREAL;
END_VAR
ConvertRadiansToDegrees := radiand * 180 / PI;
END_METHOD

METHOD GetRandomValue : LREAL
VAR_INPUT
	seed : INT;
END_VAR
_Random(Seed := seed, Num => GetRandomValue);
END_METHOD

METHOD GetRandomWithDispersion : LREAL
VAR_INPUT
	baseValue : LREAL;
	dispersion : LREAL;	
END_VAR
GetRandomWithDispersion := baseValue - dispersion + (dispersion * 2 * MathHelper.GetRandomValue(0));
END_METHOD

METHOD GetRandomWithDispersionEx : LREAL
VAR_INPUT
	minValue : LREAL;
	baseValue : LREAL;
	maxValue : LREAL;
	dispersion : LREAL;	
END_VAR
GetRandomWithDispersionEx := baseValue - dispersion + (dispersion * 2 * MathHelper.GetRandomValue(0));

IF GetRandomWithDispersionEx < minValue THEN
	GetRandomWithDispersionEx := minValue;
ELSIF GetRandomWithDispersionEx > maxValue THEN
	GetRandomWithDispersionEx := maxValue;
END_IF
END_METHOD

METHOD Truncate : LREAL
VAR_INPUT
	value : LREAL;
	precission : BYTE;
END_VAR
VAR 
	i : INT;
	factor : LREAL := 1;
END_VAR
FOR i := 1 TO precission DO
	factor := factor * 10;
END_FOR

Truncate := TO_LREAL(TRUNC(value * factor)) / factor;
END_METHOD

END_PROGRAM

// ---- Primitives/AnyType/AnyTypeHelper.TcPOU
PROGRAM AnyTypeHelper

METHOD GetAnyDescriptorByVariable : __SYSTEM.AnyType
VAR_INPUT
	variable : ANY;
END_VAR
GetAnyDescriptorByVariable := variable;
END_METHOD

END_PROGRAM

// ---- Primitives/Bit/BitHelper.TcPOU
PROGRAM BitHelper

METHOD GetBitsFromByte : BYTE
VAR_INPUT
	OriginalByte : BYTE;
	FirstBitIndex : BYTE;
	LastBitIndex : BYTE;
END_VAR
VAR
	SHLBits: BYTE;
	SHRBits: BYTE;
END_VAR
IF FirstBitIndex >= 7 OR LastBitIndex >= 7 THEN
	GetBitsFromByte := 0;
	RETURN;
END_IF;

SHLBits:= 7- LastBitIndex;
SHRBits:= FirstBitIndex + LastBitIndex;

IF SHLBits > 0 THEN
	GetBitsFromByte := SHL(OriginalByte, SHLBits);
END_IF;

IF SHRBits > 0 THEN
	GetBitsFromByte := SHR(OriginalByte, SHRBits);
END_IF;
END_METHOD

METHOD GetBitsFromDWord : DWORD
VAR_INPUT
	OriginalDword : DWORD;
	FirstBitIndex : BYTE;
	LastBitIndex : BYTE;
END_VAR
VAR
	SHLBits: BYTE;
	SHRBits: BYTE;
END_VAR
IF FirstBitIndex >= 31 OR LastBitIndex >= 31 THEN
	GetBitsFromDWord := 0;
	RETURN;
END_IF;

SHLBits:= 31 - LastBitIndex;
SHRBits:= FirstBitIndex + LastBitIndex;

IF SHLBits > 0 THEN
	GetBitsFromDWord := SHL(OriginalDword, SHLBits);
END_IF;

IF SHRBits > 0 THEN
	GetBitsFromDWord := SHR(OriginalDword, SHRBits);
END_IF;
END_METHOD

METHOD GetBitsFromLReal : LREAL
VAR_INPUT
	OriginalLreal : LREAL;
	FirstBitIndex : BYTE;
	LastBitIndex : BYTE;
END_VAR
VAR
	SHLBits: BYTE;
	SHRBits: BYTE;
END_VAR
IF FirstBitIndex >= 63 OR LastBitIndex >= 63 THEN
	GetBitsFromLReal := 0;
	RETURN;
END_IF;

SHLBits := 63 - LastBitIndex;
SHRBits := FirstBitIndex + LastBitIndex;

IF SHLBits > 0 THEN
	GetBitsFromLReal := SHL(LREAL_TO_DWORD(OriginalLreal), SHLBits);
END_IF;

IF SHRBits > 0 THEN
	GetBitsFromLReal := SHR(LREAL_TO_DWORD(OriginalLreal), SHRBits);
END_IF;
END_METHOD

METHOD GetBitsFromWord : WORD
VAR_INPUT
	OriginalWord : WORD;
	FirstBitIndex : BYTE;
	Count : BYTE;
END_VAR
VAR
	SHLBits: BYTE;
	SHRBits: BYTE;
END_VAR
IF FirstBitIndex >= 15 OR Count > 16 THEN
	GetBitsFromWord := 0;
	RETURN;
END_IF;

SHLBits:= 16 - FirstBitIndex- Count;
SHRBits:= SHLBits +FirstBitIndex ;
GetBitsFromWord := OriginalWord;

IF SHLBits > 0 THEN
	GetBitsFromWord := SHL(GetBitsFromWord, SHLBits);
END_IF;

IF SHRBits > 0 THEN
	GetBitsFromWord := SHR(GetBitsFromWord, SHRBits);
END_IF;
END_METHOD

END_PROGRAM

// ---- Primitives/Byte/ByteHelper.TcPOU
PROGRAM ByteHelper

METHOD SearchByte : DINT
VAR_INPUT
	startAddress : POINTER TO BYTE;
	startIndex : DINT;
	totalBytesCount : DINT;
	searchingByte : BYTE;
END_VAR
VAR
	i : DINT;
END_VAR
SearchByte := -1;

FOR i := startIndex TO startIndex + totalBytesCount - 1 DO
	IF startAddress[i] = searchingByte THEN
		SearchByte := i;
		RETURN;
	END_IF
END_FOR
END_METHOD

METHOD Swap2Bytes
VAR_INPUT
	data : POINTER TO ARRAY [0..1] OF BYTE;
END_VAR
VAR
	buffer : BYTE;
END_VAR
buffer := data^[0];
data^[0] := data^[1];
data^[1] := buffer;
END_METHOD

METHOD Swap4Bytes
VAR_INPUT
	data : POINTER TO ARRAY [0..3] OF BYTE;
END_VAR
VAR
	buffer : BYTE;
END_VAR
buffer := data^[0];
data^[0] := data^[3];
data^[3] := buffer;

buffer := data^[1];
data^[1] := data^[2];
data^[2] := buffer;
END_METHOD

METHOD Swap8Bytes
VAR_INPUT
	data : POINTER TO ARRAY [0..7] OF BYTE;
END_VAR
VAR
	buffer : BYTE;
END_VAR
buffer := data^[0];
data^[0] := data^[7];
data^[7] := buffer;

buffer := data^[1];
data^[1] := data^[6];
data^[6] := buffer;

buffer := data^[2];
data^[2] := data^[5];
data^[5] := buffer;

buffer := data^[3];
data^[3] := data^[4];
data^[4] := buffer;
END_METHOD

METHOD TrimBytesLeft
VAR_INPUT
	startAddress : PVOID;
	trimBytesCount : DINT; 	
END_VAR
VAR_IN_OUT
	totalBytesCount : DINT;
END_VAR
IF trimBytesCount > 0 AND trimBytesCount <= totalBytesCount THEN
	TC2_SYSTEM.MEMCPY(startAddress, startAddress + DINT_TO_UDINT(trimBytesCount), DINT_TO_UDINT(totalBytesCount - trimBytesCount));
	totalBytesCount	:= totalBytesCount - trimBytesCount;
END_IF
END_METHOD

END_PROGRAM

// ---- Timers/Timer.TcPOU
{attribute 'no_explicit_call' := 'do not call this function block directly'} 
// The wrapper around Tc2_Standard.TON
FUNCTION_BLOCK FINAL Timer EXTENDS Object IMPLEMENTS IAction
VAR
	{attribute 'OPC.UA.DA' := '0'}
	_ClassName : STRING := __POUNAME();

	{attribute 'OPC.UA.DA' := '0'}
	_Timer : Tc2_Standard.TON;
	
	{attribute 'OPC.UA.DA' := '0'}
	_PrevTimerQ : BOOL;
	{attribute 'OPC.UA.DA' := '0'}
	_Error : BOOL;
END_VAR

{attribute 'monitoring' := 'call'}
{attribute 'OPC.UA.DA.Property' := '1'}
{attribute 'OPC.UA.DA.Access' := '1'}
PROPERTY Busy : BOOL
GET
Busy := _Timer.IN AND_THEN NOT _Timer.Q;
END_GET
END_PROPERTY

{attribute 'monitoring' := 'call'}
PROPERTY ClassName : STRING
GET
ClassName := _ClassName;
END_GET
END_PROPERTY

{attribute 'monitoring' := 'call'}
{attribute 'OPC.UA.DA.Property' := '1'}
{attribute 'OPC.UA.DA.Access' := '1'}
// Timer elapsed
PROPERTY Done : BOOL
GET
Done := _Timer.Q;
END_GET
END_PROPERTY

{attribute 'monitoring' := 'call'}
{attribute 'OPC.UA.DA.Property' := '1'}
{attribute 'OPC.UA.DA.Access' := '1'}
PROPERTY ElapsedTime : TIME
GET
ElapsedTime := _Timer.ET;
END_GET
END_PROPERTY

{attribute 'monitoring' := 'call'}
{attribute 'OPC.UA.DA.Property' := '1'}
{attribute 'OPC.UA.DA.Access' := '1'}
PROPERTY Error : BOOL
GET
Error := _Error;
END_GET
END_PROPERTY

METHOD Execute
_PrevTimerQ := _Timer.Q;

_Timer();
END_METHOD

{attribute 'monitoring' := 'call'}
{attribute 'OPC.UA.DA.Property' := '1'}
{attribute 'OPC.UA.DA.Access' := '1'}
PROPERTY Interval : TIME
GET
Interval := _Timer.PT;
END_GET
SET
_Timer.PT := Interval;
END_SET
END_PROPERTY

// Restart timer if already started
METHOD Start
VAR
	//exceptionFactory : ExceptionFactory(__POUNAME(), ClassName, CurrentNamespace.Name);
END_VAR
IF _Timer.PT > T#0S THEN
	_Error := FALSE;
	
	IF _Timer.IN THEN
		_Timer(IN := FALSE);
	END_IF
	
	_Timer(IN := TRUE);
ELSE
	//exceptionFactory.ThrowException(__POSITION(), "Timer interval is not specified");
	
	_Error := TRUE;
END_IF
END_METHOD

{attribute 'monitoring' := 'call'}
{attribute 'OPC.UA.DA.Property' := '1'}
{attribute 'OPC.UA.DA.Access' := '1'}
PROPERTY Started : BOOL
GET
Started := _Timer.IN;
END_GET
END_PROPERTY

METHOD Stop
_Timer(IN := FALSE);
_Error := FALSE;
END_METHOD

// True if timer just elapsed
PROPERTY Triggered : BOOL
GET
Triggered := NOT _PrevTimerQ AND_THEN _Timer.Q;
END_GET
END_PROPERTY

END_FUNCTION_BLOCK
